(* CoDeSys 2.3.9.41 project: testApp.pro *)
(* Libraries: Util.lib 18.5.10 15:14:28, STANDARD.LIB 4.10.05 11:14:46, IECSFC.LIB 13.4.06 15:51:28, SYSLIBTIME.LIB 6.11.19 15:29:28, ANALYZATION.LIB 5.10.99 09:05:06 *)

(* PLC configuration (modules and I/O channels)
Fast discrete inputs [I_SIMPLE_INPUT] node 0, in %IB0 out %QB0 {Filtrationtime = 10}
  AT %IX0.0 [BitInput] Discrete input 1
  AT %IX0.1 [BitInput] Discrete input 2
  AT %IX0.2 [BitInput] Discrete input 3
  AT %IX0.3 [BitInput] Discrete input 4
Discrete inputs [ID130] node 1, in %IB1 out %QB1 {Filtrationtime_GeneralINP = 10; Visibility = No; PinCount = 12}
  AT %IB1.0 [ByteInput] 8 discrete inputs
  AT %IB1.1 [ByteInput] 4 discrete inputs
AT %QB2.0 [ByteOutput] 8 discrete outputs
AT %QB2.1 [ByteOutput] 4 discrete outputs
Fast analog inputs [ID125] node 3, in %IB3 out %QB3 {Flt_Comm = 50Hz 2Por}
  AT %IR3.0 [FloatInputP] AI #1 {AIN_TYPE = 4-20 mA; Peak_Filtr = 200; Flt_Ch = Off; TauRC = 10; MinFV = 0; MaxFV = 20000.0}
  AT %IR3.1 [FloatInputP] AI #2 {AIN_TYPE = 4-20 mA; Peak_Filtr = 200; Flt_Ch = Off; TauRC = 10; MinFV = 0; MaxFV = 20000.0}
  AT %IR3.2 [FloatInputP] AI #3 {AIN_TYPE = 4-20 mA; Peak_Filtr = 200; Flt_Ch = Off; TauRC = 10; MinFV = 0; MaxFV = 20000.0}
  AT %IR3.3 [FloatInputP] AI #4 {AIN_TYPE = 4-20 mA; Peak_Filtr = 200; Flt_Ch = Off; TauRC = 10; MinFV = 0; MaxFV = 20000.0}
  AT %IR3.4 [FloatInputP] AI #5 {AIN_TYPE = 4-20 mA; Peak_Filtr = 200; Flt_Ch = Off; TauRC = 10; MinFV = 0; MaxFV = 20000.0}
  AT %IR3.5 [FloatInputP] AI #6 {AIN_TYPE = 4-20 mA; Peak_Filtr = 200; Flt_Ch = Off; TauRC = 10; MinFV = 0; MaxFV = 20000.0}
  AT %IR3.6 [FloatInputP] AI #7 {AIN_TYPE = 4-20 mA; Peak_Filtr = 200; Flt_Ch = Off; TauRC = 10; MinFV = 0; MaxFV = 20000.0}
  AT %IR3.7 [FloatInputP] AI #8 {AIN_TYPE = 4-20 mA; Peak_Filtr = 200; Flt_Ch = Off; TauRC = 10; MinFV = 0; MaxFV = 20000.0}
  AT %IW3.8 [WordInput] AI read time (10ms)
Analog outputs [ID126] node 4, in %IB4 out %QB4
  AT %QR4.0 [FloatOutputP] AO #1 {AOUT_TYPE = 4-20 mA; SafeValueREAL = 0.0}
  AT %QR4.1 [FloatOutputP] AO #2 {AOUT_TYPE = 4-20 mA; SafeValueREAL = 0.0}
  AT %QR4.2 [FloatOutputP] AO #3 {AOUT_TYPE = 4-20 mA; SafeValueREAL = 0.0}
  AT %QR4.3 [FloatOutputP] AO #4 {AOUT_TYPE = 4-20 mA; SafeValueREAL = 0.0}
Special input [ID103] node 5, in %IB5 out %QB5 {Filtrationtime = 1000; PinCount = 1; WatchDogPeriod = 400; PollPeriod = 3000; Visibility = No}
  AT %IX5.0 [BitInput] Special input
Special output [ID104] node 6, in %IB6 out %QB6 {Visibility = No; PinCount = 1}
  AT %QX6.0 [BitOutput] Special output
*)

(* POU PLC_PRG, CFC *)
PROGRAM PLC_PRG
VAR
	blink_0: BLINK;
END_VAR
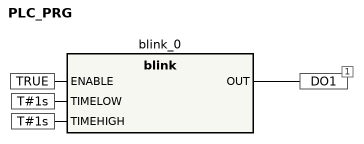
_CFC_ (* Continuous Function Chart, elements in execution order *)
#0 blink_0:blink(ENABLE: TRUE, TIMELOW: T#1s, TIMEHIGH: T#1s)
#1 DO1 <= #0.OUT
_END_CFC_
(* the same logic as Structured Text *)
blink_0(ENABLE := TRUE, TIMELOW := T#1s, TIMEHIGH := T#1s);
DO1 := blink_0.OUT;
END_PROGRAM
